{attribute 'GeneratedUsingTerminal: EL3208-0000-0017'}
{attribute addProperty BoxType "EL3208-0000-0017"}
{attribute addProperty Id "RTD_Inputs_Channel_1AT %I*RTD_Inputs_Channel_9575FEA17RTD_Inputs_Channel_2AT %I*RTD_Inputs_Channel_9575FEA17RTD_Inputs_Channel_3AT %I*RTD_Inputs_Channel_9575FEA17RTD_Inputs_Channel_4AT %I*RTD_Inputs_Channel_9575FEA17RTD_Inputs_Channel_5AT %I*RTD_Inputs_Channel_9575FEA17RTD_Inputs_Channel_6AT %I*RTD_Inputs_Channel_9575FEA17RTD_Inputs_Channel_7AT %I*RTD_Inputs_Channel_9575FEA17RTD_Inputs_Channel_8AT %I*RTD_Inputs_Channel_9575FEA17WcStateAT %I*WcState_9091E0EB2InfoDataAT %I*InfoData_94A18F5E2"}
{attribute addProperty CRC "2169660232"}
{attribute addProperty Size "60"}
TYPE EL3208_81526348 EXTENDS EtcSlaveTerminalBase_947E5A46 :
STRUCT
	{attribute addProperty Name "RTD_Inputs_Channel_1"}
	RTD_Inputs_Channel_1 : RTD_Inputs_Channel_9575FEA1;
	{attribute addProperty Name "RTD_Inputs_Channel_2"}
	RTD_Inputs_Channel_2 : RTD_Inputs_Channel_9575FEA1;
	{attribute addProperty Name "RTD_Inputs_Channel_3"}
	RTD_Inputs_Channel_3 : RTD_Inputs_Channel_9575FEA1;
	{attribute addProperty Name "RTD_Inputs_Channel_4"}
	RTD_Inputs_Channel_4 : RTD_Inputs_Channel_9575FEA1;
	{attribute addProperty Name "RTD_Inputs_Channel_5"}
	RTD_Inputs_Channel_5 : RTD_Inputs_Channel_9575FEA1;
	{attribute addProperty Name "RTD_Inputs_Channel_6"}
	RTD_Inputs_Channel_6 : RTD_Inputs_Channel_9575FEA1;
	{attribute addProperty Name "RTD_Inputs_Channel_7"}
	RTD_Inputs_Channel_7 : RTD_Inputs_Channel_9575FEA1;
	{attribute addProperty Name "RTD_Inputs_Channel_8"}
	RTD_Inputs_Channel_8 : RTD_Inputs_Channel_9575FEA1;
	{attribute addProperty Name "WcState"}
	WcState : WcState_9091E0EB;
	{attribute addProperty Name "InfoData"}
	InfoData : InfoData_94A18F5E;
END_STRUCT
END_TYPE

(* stored: Version 1.2.0.0, ProductVersion 3.1.4024.9
   DUT EL3208_81526348: Id {67b7d185-9b2e-4040-ac75-fd22367cea8a} *)
